% RSLogix 500 project STRING CTRL LOGIC PRACTICE.RSS, saved by version 8.30.00.16 %
PROJECT "SIM_PLC"    % processor: Bul.1763 MicroLogix 1100 Series B %

PROGRAM FILES
  LAD 2 "MAIN"  4 rungs
  LAD 3 "INPUTS"  2 rungs
  LAD 4 "STR SCAN"  2 rungs
  LAD 5 "INV MGMT"  7 rungs

DATA FILES
  O0 OUTPUT  4 elements
  I1 INPUT  6 elements
  S2 STATUS  66 elements
  B3 BINARY  1 elements
  T4 TIMER  1 elements
  C5 COUNTER  1 elements
  R6 CONTROL  1 elements
  N7 INTEGER  10 elements
  F8 FLOAT  1 elements
  ST9 STRING  9 elements

LADDER 2 "MAIN"
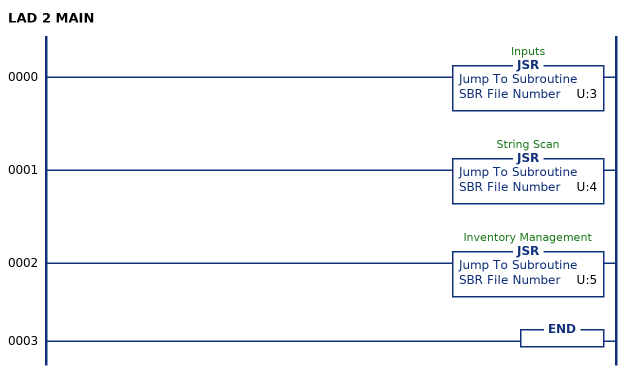
% Rung: 0 %
SOR JSR U:3 EOR
%   U:3  "Inputs" %
% Rung: 1 %
SOR JSR U:4 EOR
%   U:4  "String Scan" %
% Rung: 2 %
SOR JSR U:5 EOR
%   U:5  "Inventory Management" %
% Rung: 3 %
SOR END EOR

LADDER 3 "INPUTS"
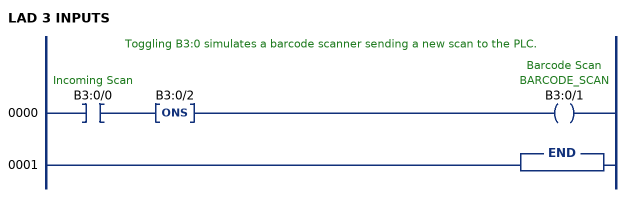
% Rung: 0 %  % edit flag set %
% Toggling B3:0 simulates a barcode scanner sending a new scan to the PLC. %
SOR XIC B3:0/0 ONS B3:0/2 OTE B3:0/1 EOR
%   B3:0/0  "Incoming Scan" %
%   B3:0/1  BARCODE_SCAN  "Barcode Scan" %
% Rung: 1 %
SOR END EOR

LADDER 4 "STR SCAN"
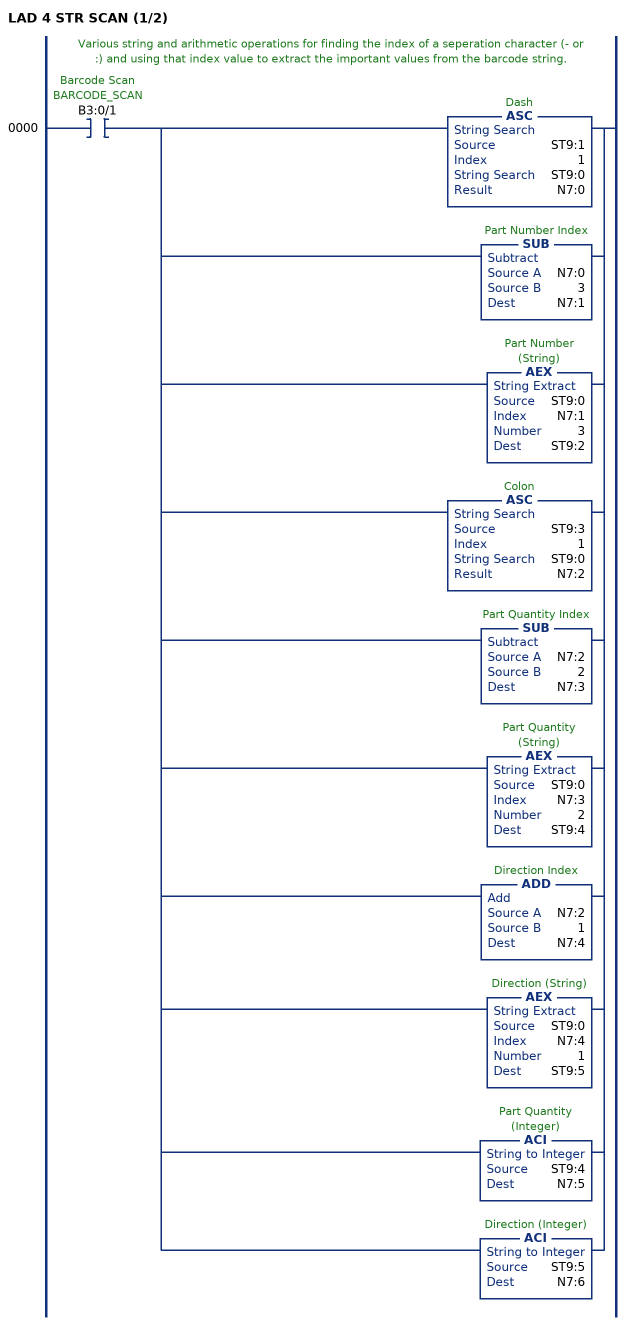
% Rung: 0 %  % edit flag set %
% Various string and arithmetic operations for finding the index of a seperation character (- or :) and using that index value to extract the important values from the barcode string. %
SOR XIC B3:0/1 BST ASC ST9:1 1 ST9:0 N7:0 NXB SUB N7:0 3 N7:1 NXB AEX ST9:0 N7:1 3 ST9:2 NXB ASC ST9:3 1 ST9:0 N7:2 NXB SUB N7:2 2 N7:3 NXB AEX ST9:0 N7:3 2 ST9:4 NXB ADD N7:2 1 N7:4 NXB AEX ST9:0 N7:4 1 ST9:5 NXB ACI ST9:4 N7:5 NXB ACI ST9:5 N7:6 BND EOR
%   B3:0/1  BARCODE_SCAN  "Barcode Scan" %
%   ST9:1  "Dash" %
%   ST9:0  "Barcode String" %
%   N7:0  "Dash Index" %
%   N7:1  "Part Number Index" %
%   ST9:2  "Part Number (String)" %
%   ST9:3  "Colon" %
%   N7:2  "Colon Index" %
%   N7:3  "Part Quantity Index" %
%   ST9:4  "Part Quantity (String)" %
%   N7:4  "Direction Index" %
%   ST9:5  "Direction (String)" %
%   N7:5  "Part Quantity (Integer)" %
%   N7:6  "Direction (Integer)" %

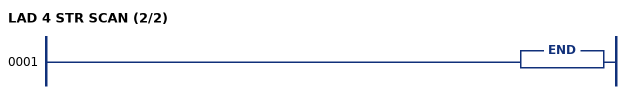
% Rung: 1 %
SOR END EOR

LADDER 5 "INV MGMT"
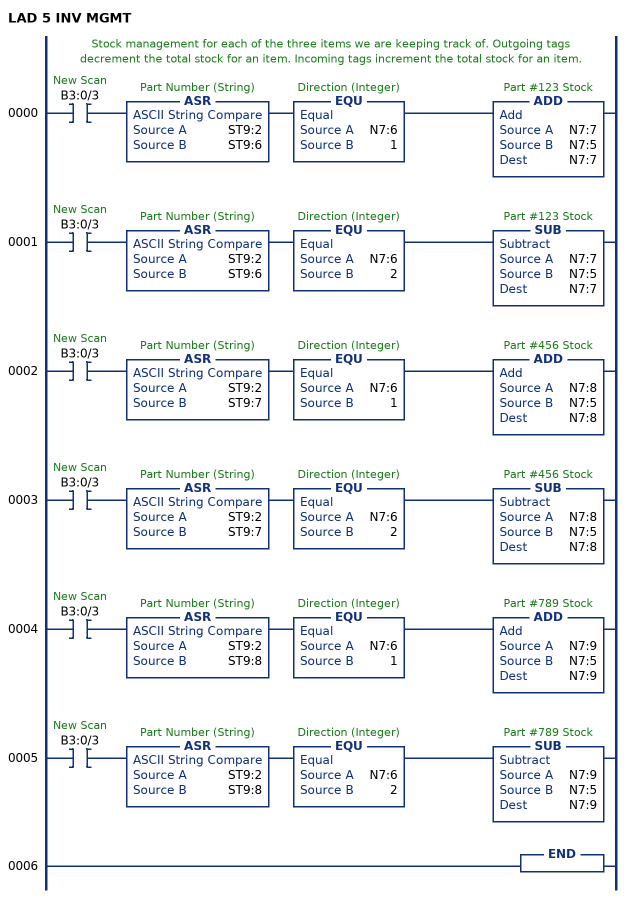
% Rung: 0 %
% Stock management for each of the three items we are keeping track of. Outgoing tags decrement the total stock for an item. Incoming tags increment the total stock for an item. %
SOR XIC B3:0/3 ASR ST9:2 ST9:6 EQU N7:6 1 ADD N7:7 N7:5 N7:7 EOR
%   B3:0/3  "New Scan" %
%   ST9:2  "Part Number (String)" %
%   ST9:6  "Part #123" %
%   N7:6  "Direction (Integer)" %
%   N7:7  "Part #123 Stock" %
%   N7:5  "Part Quantity (Integer)" %
% Rung: 1 %
SOR XIC B3:0/3 ASR ST9:2 ST9:6 EQU N7:6 2 SUB N7:7 N7:5 N7:7 EOR
%   B3:0/3  "New Scan" %
%   ST9:2  "Part Number (String)" %
%   ST9:6  "Part #123" %
%   N7:6  "Direction (Integer)" %
%   N7:7  "Part #123 Stock" %
%   N7:5  "Part Quantity (Integer)" %
% Rung: 2 %
SOR XIC B3:0/3 ASR ST9:2 ST9:7 EQU N7:6 1 ADD N7:8 N7:5 N7:8 EOR
%   B3:0/3  "New Scan" %
%   ST9:2  "Part Number (String)" %
%   ST9:7  "Part #456" %
%   N7:6  "Direction (Integer)" %
%   N7:8  "Part #456 Stock" %
%   N7:5  "Part Quantity (Integer)" %
% Rung: 3 %
SOR XIC B3:0/3 ASR ST9:2 ST9:7 EQU N7:6 2 SUB N7:8 N7:5 N7:8 EOR
%   B3:0/3  "New Scan" %
%   ST9:2  "Part Number (String)" %
%   ST9:7  "Part #456" %
%   N7:6  "Direction (Integer)" %
%   N7:8  "Part #456 Stock" %
%   N7:5  "Part Quantity (Integer)" %
% Rung: 4 %
SOR XIC B3:0/3 ASR ST9:2 ST9:8 EQU N7:6 1 ADD N7:9 N7:5 N7:9 EOR
%   B3:0/3  "New Scan" %
%   ST9:2  "Part Number (String)" %
%   ST9:8  "Part #789" %
%   N7:6  "Direction (Integer)" %
%   N7:9  "Part #789 Stock" %
%   N7:5  "Part Quantity (Integer)" %
% Rung: 5 %
SOR XIC B3:0/3 ASR ST9:2 ST9:8 EQU N7:6 2 SUB N7:9 N7:5 N7:9 EOR
%   B3:0/3  "New Scan" %
%   ST9:2  "Part Number (String)" %
%   ST9:8  "Part #789" %
%   N7:6  "Direction (Integer)" %
%   N7:9  "Part #789 Stock" %
%   N7:5  "Part Quantity (Integer)" %
% Rung: 6 %
SOR END EOR
